Yaskawa INFORM job: LTESRCS1.JBI

/JOB
//NAME LTESRCS1
//POS
///NPOS 0,0,0,0,0,0
//INST
///DATE 2019/11/21 19:10
///ATTR SC,RW,MC
///GROUP1 RB1,BS1
///GROUP2 ST1
///LVARS 2,0,0,0,0,0,0,0
NOP
GETARG LB000 IARG#(1)
GETARG LB001 IARG#(2)
JUMP *END IF LB000<>1
SKILLSND ATTR=3 "LSRCHED LT:1"
*END
END
